ABB RAPID module: Point_ALL.mod

MODULE Point_ALL

    !************************************************************************************************!
    CONST robtarget Point_home:=[[377.25,-367.22,182.16],[0,0.986757,0.162205,0],[-1,-1,0,0],[9E+09,9E+09,9E+09,9E+09,9E+09,9E+09]];
    CONST robtarget Point_SafeHigh:=[[377.24,-367.23,182.16],[0,0.986763,0.162169,0],[-1,-1,0,0],[9E+09,9E+09,9E+09,9E+09,9E+09,9E+09]];
    CONST robtarget Point_Pick1:=[[424.80,-201.45,131.11],[0,0.988408,0.151822,0],[-1,0,0,0],[9E+09,9E+09,9E+09,9E+09,9E+09,9E+09]];
    CONST robtarget Point_Pick2:=[[359.67,-200.70,131.03],[0,0.988788,0.149324,0],[-1,0,0,0],[9E+09,9E+09,9E+09,9E+09,9E+09,9E+09]];
    CONST robtarget Point_Over1:=[[392.27,-225.61,161.55],[0,0.986741,0.162301,0],[-1,0,0,0],[9E+09,9E+09,9E+09,9E+09,9E+09,9E+09]];
    CONST robtarget Point_Over2:=[[328.99,-470.77,161.55],[0,0.986744,0.162284,0],[-1,-1,0,0],[9E+09,9E+09,9E+09,9E+09,9E+09,9E+09]];
    CONST robtarget Point_Snap:=[[328.78,-557.91,106.7],[0,0.986756,0.162214,0],[-1,-1,0,0],[9E+09,9E+09,9E+09,9E+09,9E+09,9E+09]];
    CONST robtarget Point_Snap1:=[[328.78,-557.91,106.7],[0,0.986756,0.162214,0],[-1,-1,0,0],[9E+09,9E+09,9E+09,9E+09,9E+09,9E+09]];
    CONST robtarget Point_Snap2:=[[328.78,-557.91,106.7],[0,0.986756,0.162214,0],[-1,-1,0,0],[9E+09,9E+09,9E+09,9E+09,9E+09,9E+09]];
    CONST robtarget Point_Put1:=[[328.78,-557.91,106.7],[0,0.986756,0.162214,0],[-1,-1,0,0],[9E+09,9E+09,9E+09,9E+09,9E+09,9E+09]];
    CONST robtarget Point_Put2:=[[328.78,-557.91,106.7],[0,0.986756,0.162214,0],[-1,-1,0,0],[9E+09,9E+09,9E+09,9E+09,9E+09,9E+09]];
    CONST robtarget Point_Quliao1:=[[328.78,-557.91,106.7],[0,0.986756,0.162214,0],[-1,-1,0,0],[9E+09,9E+09,9E+09,9E+09,9E+09,9E+09]];
    CONST robtarget Point_Quliao2:=[[328.78,-557.91,106.7],[0,0.986756,0.162214,0],[-1,-1,0,0],[9E+09,9E+09,9E+09,9E+09,9E+09,9E+09]];
    CONST robtarget Guodu1:=[[328.78,-557.91,106.7],[0,0.986756,0.162214,0],[-1,-1,0,0],[9E+09,9E+09,9E+09,9E+09,9E+09,9E+09]];
    CONST robtarget Guodu2:=[[328.78,-557.91,106.7],[0,0.986756,0.162214,0],[-1,-1,0,0],[9E+09,9E+09,9E+09,9E+09,9E+09,9E+09]];
    CONST robtarget Guodu3:=[[328.78,-557.91,106.7],[0,0.986756,0.162214,0],[-1,-1,0,0],[9E+09,9E+09,9E+09,9E+09,9E+09,9E+09]];
    CONST robtarget Guodu4:=[[328.78,-557.91,106.7],[0,0.986756,0.162214,0],[-1,-1,0,0],[9E+09,9E+09,9E+09,9E+09,9E+09,9E+09]];
    CONST robtarget Point_Assemble1:=[[328.78,-557.91,106.17],[0,0.986754,0.162226,0],[-1,-1,0,0],[9E+09,9E+09,9E+09,9E+09,9E+09,9E+09]];
    CONST robtarget Point_Assemble2:=[[328.78,-557.91,106.17],[0,0.986754,0.162226,0],[-1,-1,0,0],[9E+09,9E+09,9E+09,9E+09,9E+09,9E+09]];
    CONST robtarget Point_Throw1:=[[324.13,-400.34,144.94],[0,0.986684,0.162651,0],[-1,-1,0,0],[9E+09,9E+09,9E+09,9E+09,9E+09,9E+09]];
    CONST robtarget Point_Throw2:=[[324.13,-400.34,144.94],[0,0.986684,0.162651,0],[-1,-1,0,0],[9E+09,9E+09,9E+09,9E+09,9E+09,9E+09]];
    CONST robtarget Point_Pallet0:=[[192,-350.56,83],[0,0.730241,-0.68319,0],[-1,-1,0,1],[9E+09,9E+09,9E+09,9E+09,9E+09,9E+09]];
    CONST robtarget Point_Pallet1:=[[311.16,-353.26,83],[0,0.730241,-0.68319,0],[-1,0,0,1],[9E+09,9E+09,9E+09,9E+09,9E+09,9E+09]];
    CONST robtarget Point_Pallet2:=[[192,-208.26,83],[0,0.730241,-0.68319,0],[0,-1,0,1],[9E+09,9E+09,9E+09,9E+09,9E+09,9E+09]];
ENDMODULE
